Yaskawa INFORM job: X2_22-23(-90,180).JBI

/JOB
//NAME X2_22-23(-90,180)
///FOLDERNAME X2
//POS
///NPOS 121,121,119,9,0,0
///TOOL 0
///POSTYPE PULSE
///PULSE
C00000=-2000,-95440,-72516,0,38121,0
C00001=80443,-95440,-72516,46202,38121,-50067
C00002=121048,-35889,-42121,1043,37047,-65138
C00003=121557,-2539,-17456,-43794,56524,-32797
C00004=120863,2743,-10296,-44250,54945,-32361
C00005=120596,4906,-7348,-44467,54301,-32168
C00006=120755,7039,-5502,-44562,54352,-32106
C00007=120722,6457,-5983,-44548,54334,-32114
C00008=120719,6604,-4609,-44933,53775,-31814
C00009=120722,6457,-5983,-44548,54334,-32114
C00010=120988,4291,-8953,-44325,54985,-32311
C00011=121680,-993,-16157,-43855,56581,-32759
C00012=120048,-2169,-23700,-17577,56183,-40243
C00013=120438,2634,-16754,-18201,54544,-39794
C00014=120588,4602,-13901,-18464,53869,-39607
C00015=120747,6727,-12066,-18575,53869,-39539
C00016=120731,6185,-12507,-18566,53858,-39544
C00017=120727,6181,-11266,-18742,53130,-39409
C00018=120731,6185,-12507,-18566,53858,-39544
C00019=120584,4213,-15378,-18303,54543,-39732
C00020=120201,-590,-22366,-17676,56206,-40184
C00021=120684,5680,-12751,-24181,58802,-41191
C00022=120685,5691,-12742,-24181,58802,-41191
C00023=120646,5363,-16101,-23722,60533,-41605
C00024=120645,1544,-17222,-24010,59364,-41338
C00025=120685,5695,-12739,-24181,58802,-41191
C00026=120685,5705,-12730,-24145,60239,-39557
C00027=120685,5848,-12606,-24145,60236,-39557
C00028=120407,6153,-6117,-43461,53553,-40856
C00029=120685,5980,-7491,-43224,54249,-41062
C00030=120685,5834,-10671,-42343,55652,-41764
C00031=121048,-35889,-42121,1043,37047,-65138
C00032=80443,-95440,-72516,46202,38121,-50067
C00033=628,-74499,-67639,57475,89722,-72456
C00034=628,-74499,-67639,57475,89722,-72456
C00035=57022,-39792,-97587,14580,73098,-62715
C00036=77807,6055,-39746,10148,68442,-55630
C00037=79243,8316,-34713,9405,66379,-55331
C00038=80169,10516,-31635,8886,65529,-55089
C00039=80963,12031,-30280,8399,65395,-54832
C00040=80889,11723,-30556,8444,65413,-54856
C00041=80889,11351,-30020,8477,64899,-54893
C00042=80459,11155,-31041,8710,65464,-54995
C00043=79913,10174,-33131,8996,66291,-55115
C00044=78505,7891,-38206,9727,68362,-55410
C00045=77753,5785,-39720,10191,68296,-55659
C00046=79192,8060,-34680,9447,66235,-55360
C00047=82054,8043,-33590,7724,65287,-54470
C00048=82379,9432,-32364,7521,65217,-54367
C00049=82297,9081,-32674,7571,65235,-54393
C00050=82297,8847,-32336,7591,64909,-54415
C00051=80432,10909,-31095,8733,65375,-55011
C00052=79885,9924,-33187,9019,66201,-55131
C00053=78475,7632,-38265,9751,68270,-55428
C00054=83648,6461,-36170,1745,63660,-53011
C00055=83747,5652,-35361,1694,62744,-52991
C00056=84187,6753,-32863,1416,61768,-52855
C00057=81142,10477,-29433,3447,61652,-53915
C00058=80255,9791,-30406,4031,61937,-54214
C00059=80258,11096,-32246,3966,63735,-54150
C00060=57022,-39792,-97587,14580,73098,-62715
C00061=628,-74499,-67639,57475,89722,-72456
C00062=628,-74499,-67639,57475,89722,-72456
C00063=628,-74499,-67639,57475,89722,-72456
C00064=628,-74499,-67639,57475,89722,-72456
C00065=71892,-109130,-85039,20754,40171,-11669
C00066=106389,-40524,-53403,24815,61142,19479
C00067=120470,1866,-17440,30101,56195,36353
C00068=120719,2683,-16651,30153,56013,36673
C00069=120773,4699,-13768,30370,55352,36490
C00070=120564,7533,-11305,30511,55374,36401
C00071=120670,6740,-11178,30619,54915,36303
C00072=120665,6751,-9510,30988,54034,36013
C00073=120670,6740,-11178,30619,54915,36303
C00074=120615,4703,-14100,30391,55587,36492
C00075=120473,-266,-21211,29878,57224,36936
C00076=121398,-1811,-23726,17127,56782,40252
C00077=120993,2938,-16799,17744,55126,39804
C00078=120837,4887,-13955,18002,54444,39619
C00079=120627,7720,-11489,18149,54432,39528
C00080=120605,6750,-11571,18262,54010,39442
C00081=120600,6748,-9914,18499,53040,39261
C00082=120605,6750,-11571,18262,54010,39442
C00083=121150,-14,-21462,17373,56384,40085
C00084=114935,6727,-10898,18108,63991,38712
C00085=105615,-2055,-15067,38715,63232,35896
C00086=105666,5748,-4871,39423,61430,35186
C00087=115774,5149,-8950,35948,58489,37624
C00088=118188,4605,-11063,30087,58489,38356
C00089=120685,6333,-7231,42675,54657,41140
C00090=120685,6258,-8528,42321,55226,41422
C00091=120685,6198,-11659,41481,56657,42109
C00092=628,-74499,-67639,57475,89722,-72456
C00093=628,-74499,-67639,57475,89722,-72456
C00094=73729,14650,-65218,39624,99784,34982
C00095=79038,5651,-41829,36469,82879,30814
C00096=79794,8712,-36062,36285,80989,30462
C00097=80238,10863,-32413,36196,79892,30261
C00098=80449,12924,-30562,36114,79745,30290
C00099=80337,12469,-30973,36158,79803,30267
C00100=80337,11828,-30094,36241,79095,30031
C00101=80425,12177,-31517,36106,79921,30344
C00102=80141,10890,-33898,36156,80684,30490
C00103=79405,7814,-39711,36325,82587,30850
C00104=79095,5770,-41687,36447,82837,30820
C00105=79848,8834,-35915,36264,80946,30468
C00106=80509,11322,-31838,36094,79692,30298
C00107=80683,12908,-30408,36027,79574,30324
C00108=80563,12412,-30857,36075,79637,30299
C00109=80563,11846,-30077,36150,79008,30090
C00110=80446,12400,-31453,36090,79975,30369
C00111=80162,11117,-33833,36141,80739,30516
C00112=79428,8050,-39643,36311,82643,30877
C00113=80369,12305,-32773,40785,82539,30314
C00114=80366,10908,-30990,40925,81149,29769
C00115=80599,11314,-29317,40908,80419,29578
C00116=80511,11265,-29307,40945,80432,29547
C00117=80326,10673,-31042,40949,81098,29733
C00118=80329,12062,-32831,40808,82488,30278
C00119=73729,14650,-65218,39624,99784,34982
C00120=-2800,-56338,-97337,367,83074,-232
BC00000=23532,523905,788952
BC00001=125909,496171,117576
BC00002=159989,496171,117576
BC00003=146377,457946,17
BC00004=146377,457946,17
BC00005=146377,457946,17
BC00006=146377,457946,17
BC00007=146377,457946,17
BC00008=146377,457946,17
BC00009=146377,457946,17
BC00010=146377,457946,17
BC00011=146377,457946,17
BC00012=124676,474529,2658
BC00013=124676,474529,2658
BC00014=124676,474529,2658
BC00015=124676,474529,2658
BC00016=124676,474529,2658
BC00017=124676,474529,2658
BC00018=124676,474529,2658
BC00019=124676,474529,2658
BC00020=124676,474529,2658
BC00021=109348,473025,40679
BC00022=109185,468237,19665
BC00023=109120,466322,11259
BC00024=109120,466322,11259
BC00025=109120,466322,11259
BC00026=113377,463743,16288
BC00027=162486,455184,17102
BC00028=158679,453956,17
BC00029=157926,455904,17
BC00030=156043,460776,17
BC00031=159989,496171,117576
BC00032=125909,496171,117576
BC00033=97158,523229,426323
BC00034=97158,523229,1005604
BC00035=48431,468399,1061681
BC00036=65052,442237,1075139
BC00037=65052,442237,1075139
BC00038=65052,442237,1075139
BC00039=65052,442237,1075139
BC00040=65052,442237,1075139
BC00041=65052,442237,1075139
BC00042=65052,442237,1075139
BC00043=65052,442237,1075139
BC00044=65052,442237,1075139
BC00045=2261,453176,1075139
BC00046=2261,453176,1075139
BC00047=2261,453176,1075139
BC00048=2261,453176,1075139
BC00049=2261,453176,1075139
BC00050=2261,453176,1075139
BC00051=2261,453176,1075139
BC00052=2261,453176,1075139
BC00053=2261,453176,1075139
BC00054=1592,459940,1075139
BC00055=1592,454468,1075139
BC00056=1592,452279,1075139
BC00057=59392,440617,1075139
BC00058=57917,442806,1075139
BC00059=58212,448278,1075139
BC00060=48431,468399,1061681
BC00061=97158,523229,1005604
BC00062=97158,523229,842352
BC00063=97158,523229,842352
BC00064=97158,523229,1051970
BC00065=250466,483638,320114
BC00066=268157,471482,125895
BC00067=279228,463874,4352
BC00068=279439,463729,2036
BC00069=279439,463729,2036
BC00070=279439,463729,2036
BC00071=279439,463729,2036
BC00072=279439,463729,2036
BC00073=279439,463729,2036
BC00074=279439,463729,2036
BC00075=279439,463729,2036
BC00076=313684,475025,18299
BC00077=313684,475025,18299
BC00078=313684,475025,18299
BC00079=313684,475025,18299
BC00080=313684,475025,18299
BC00081=313684,475025,18299
BC00082=313684,475025,18299
BC00083=313684,475025,18299
BC00084=295059,466219,85453
BC00085=298191,460141,56261
BC00086=298191,460141,56261
BC00087=322149,463189,26141
BC00088=278371,455636,25524
BC00089=279361,453981,17
BC00090=280099,455914,17
BC00091=281944,460744,17
BC00092=97158,523229,426323
BC00093=97158,523229,1033177
BC00094=194066,506419,1075139
BC00095=165051,440056,1075139
BC00096=165051,440056,1075139
BC00097=165051,440056,1075139
BC00098=165051,440056,1075139
BC00099=165051,440056,1075139
BC00100=165051,440056,1075139
BC00101=165051,440056,1075139
BC00102=165051,440056,1075139
BC00103=165051,440056,1075139
BC00104=226024,450581,1075139
BC00105=226024,450581,1075139
BC00106=226024,450581,1075139
BC00107=226024,450581,1075139
BC00108=226024,450581,1075139
BC00109=226024,450581,1075139
BC00110=226024,450581,1075139
BC00111=226024,450581,1075139
BC00112=226024,450581,1075139
BC00113=238899,457644,1075139
BC00114=239227,452207,1075139
BC00115=239359,450033,1075139
BC00116=172415,438485,1075139
BC00117=172284,440660,1075139
BC00118=171955,446096,1075139
BC00119=194066,506419,1075139
BC00120=194066,523905,1075139
EC00000=798156,-1296783
EC00001=798156,-1296783
EC00002=798156,-1296783
EC00003=798156,-1296783
EC00004=798156,-1296783
EC00005=798156,-1296783
EC00006=798156,-1296783
EC00007=798156,-1296783
EC00008=798156,-1296783
EC00009=798156,-1296783
EC00010=798156,-1296783
EC00011=798156,-1296783
EC00012=798156,-1296783
EC00013=798156,-1296783
EC00014=798156,-1296783
EC00015=798156,-1296783
EC00016=798156,-1296783
EC00017=798156,-1296783
EC00018=798156,-1296783
EC00019=798156,-1296783
EC00020=798156,-1296783
EC00021=798156,-1296783
EC00022=798156,-1296783
EC00023=798156,-1296783
EC00024=798156,-1296783
EC00025=798156,-1296783
EC00026=798156,-1296783
EC00027=798156,-1296783
EC00028=798156,-1296783
EC00029=798156,-1296783
EC00030=798156,-1296783
EC00031=798156,-1296783
EC00032=798156,-1296783
EC00033=798156,-1296783
EC00034=798156,-1296783
EC00035=798156,-1296783
EC00036=798156,-1296783
EC00037=798156,-1296783
EC00038=798156,-1296783
EC00039=798156,-1296783
EC00040=798156,-1296783
EC00041=798156,-1296783
EC00042=798156,-1296783
EC00043=798156,-1296783
EC00044=798156,-1296783
EC00045=798156,-1296783
EC00046=798156,-1296783
EC00047=798156,-1296783
EC00048=798156,-1296783
EC00049=798156,-1296783
EC00050=798156,-1296783
EC00051=798156,-1296783
EC00052=798156,-1296783
EC00053=798156,-1296783
EC00054=798156,-1296783
EC00055=798156,-1296783
EC00056=798156,-1296783
EC00057=798156,-1296783
EC00058=798156,-1296783
EC00059=798156,-1296783
EC00060=859390,-983133
EC00061=868219,-545682
EC00062=798156,-183832
EC00063=798156,-183832
EC00064=798156,-183832
EC00065=798156,-183832
EC00066=798156,-183832
EC00067=798156,-183832
EC00068=798156,-183832
EC00069=798156,-183832
EC00070=798156,-183832
EC00071=798156,-183832
EC00072=798156,-183832
EC00073=798156,-183832
EC00074=798156,-183832
EC00075=798156,-183832
EC00076=798156,-183832
EC00077=798156,-183832
EC00078=798156,-183832
EC00079=798156,-183832
EC00080=798156,-183832
EC00081=798156,-183832
EC00082=798156,-183832
EC00083=798156,-183832
EC00084=798156,-183832
EC00085=798156,-183832
EC00086=798156,-183832
EC00087=798156,-183832
EC00088=798156,-183832
EC00089=798156,-183832
EC00090=798156,-183832
EC00091=798156,-183832
EC00092=798156,-183832
EC00093=798156,-183832
EC00094=798156,-183832
EC00095=798156,-183832
EC00096=798156,-183832
EC00097=798156,-183832
EC00098=798156,-183832
EC00099=798156,-183832
EC00100=798156,-183832
EC00101=798156,-183832
EC00102=798156,-183832
EC00103=798156,-183832
EC00104=798156,-183832
EC00105=798156,-183832
EC00106=798156,-183832
EC00107=798156,-183832
EC00108=798156,-183832
EC00109=798156,-183832
EC00110=798156,-183832
EC00111=798156,-183832
EC00112=798156,-183832
EC00113=798156,-183832
EC00114=798156,-183832
EC00115=798156,-183832
EC00116=798156,-183832
EC00117=798156,-183832
EC00118=798156,-183832
///POSTYPE BASE
///RECTAN
///RCONF 0,0,0,0,1,0,0,0,0,0,0,0,0,0,0,0,0,0,0,0,0,0,0,0
P00006=2.006,1.622,-0.565,0.0000,0.0000,0.0000
P00021=0.073,2.058,-0.109,0.0000,0.0000,0.0000
P00022=2.006,1.622,-0.565,0.0000,0.0000,0.0000
///RCONF 0,0,0,0,0,0,0,0,0,0,0,0,0,0,0,0,0,0,0,0,0,0,0,0
P00023=-2.957,-4.083,2.762,0.0000,0.0000,0.0000
P00024=-1.466,-0.226,-0.419,0.0000,0.0000,0.0000
P00025=3.643,0.007,-2.585,0.0000,0.0000,0.0000
P00026=2.644,0.055,-2.583,0.0000,0.0000,0.0000
P00027=2.278,0.099,-4.210,0.0000,0.0000,0.0000
P00028=-1.778,-0.182,-2.050,0.0000,0.0000,0.0000
//INST
///DATE 2024/12/18 14:18
///ATTR SC,RW
///GROUP1 RB1,BS1
///GROUP2 ST1
NOP
'X2_22-23(-90,180)
MOVJ C00000 BC00000 VJ=100.00  +MOVJ EC00000 VJ=100.00
MOVJ C00001 BC00001 VJ=100.00  +MOVJ EC00001 VJ=100.00
MOVJ C00002 BC00002 VJ=100.00  +MOVJ EC00002 VJ=100.00
'Path S4216
SFTOF3D
MOVJ C00003 BC00003 VJ=100.00  +MOVJ EC00003 VJ=100.00
MOVL C00004 BC00004 V=800.0  +MOVJ EC00004 VJ=100.00
SMOVL C00005 BC00005 V=166.7  +MOVJ EC00005
SREFP 3 C00006 BC00006  +REFP EC00006
CALL JOB:SEARCH-R1-S13D
SET P022 P006
SFTON3D P022
SMOVL C00007 BC00007 V=166.7  +MOVJ EC00007
SREFP 3 C00008 BC00008  +REFP EC00008
CALL JOB:SEARCH-R1-S13D
SET P022 P006
SFTON3D P022
SMOVL C00009 BC00009 V=166.7  +MOVJ EC00009
MOVL C00010 BC00010 V=800.0  +MOVJ EC00010 VJ=100.00
MOVL C00011 BC00011 V=1000.0  +MOVJ EC00011 VJ=100.00
'EndPath S4216
'Path S3525
SFTOF3D
MOVJ C00012 BC00012 VJ=100.00  +MOVJ EC00012 VJ=100.00
MOVL C00013 BC00013 V=800.0  +MOVJ EC00013 VJ=100.00
SMOVL C00014 BC00014 V=166.7  +MOVJ EC00014
SREFP 3 C00015 BC00015  +REFP EC00015
CALL JOB:SEARCH-R1-S13D
SET P021 P006
SFTON3D P021
SMOVL C00016 BC00016 V=166.7  +MOVJ EC00016
SREFP 3 C00017 BC00017  +REFP EC00017
CALL JOB:SEARCH-R1-S13D
SET P021 P006
SFTON3D P021
SMOVL C00018 BC00018 V=166.7  +MOVJ EC00018
MOVL C00019 BC00019 V=800.0  +MOVJ EC00019 VJ=100.00
MOVL C00020 BC00020 V=1000.0  +MOVJ EC00020 VJ=100.00
'EndPath S3525
'Path W3526
SFTOF3D
SFTON3D P021
MOVJ C00021 BC00021 VJ=100.00  +MOVJ EC00021 VJ=100.00
SMOVL C00022 BC00022 V=800.0  +MOVJ EC00022
REFP 1 RB1 C00023 BC00023
REFP 2 RB1 C00024 BC00024
SMOVL C00025 BC00025 V=166.7 PL=0  +MOVJ EC00023
MACRO1 MJ#(0) ARGF18
ARCON
SMOVL C00026 BC00026 V=8.3  +MOVJ EC00024
SFTON3D P022
SMOVL C00027 BC00027 V=8.3  +MOVJ EC00025
SMOVL C00028 BC00028 V=8.3  +MOVJ EC00026
ARCOF
SMOVL C00029 BC00029 V=800.0  +MOVJ EC00027
SMOVL C00030 BC00030 V=1000.0  +MOVJ EC00028
SFTOF3D
'EndPath W3526
MOVJ C00031 BC00031 VJ=100.00  +MOVJ EC00029 VJ=100.00
MOVJ C00032 BC00032 VJ=100.00  +MOVJ EC00030 VJ=100.00
MOVJ C00033 BC00033 VJ=100.00  +MOVJ EC00031 VJ=100.00
'R-L Trip
MOVJ C00034 BC00034 VJ=100.00  +MOVJ EC00032 VJ=100.00
CALL JOB:CLEAN-R1_KM_NEW
MOVJ C00035 BC00035 VJ=100.00  +MOVJ EC00033 VJ=100.00
'Path S4217
SFTOF3D
MOVJ C00036 BC00036 VJ=100.00  +MOVJ EC00034 VJ=100.00
MOVL C00037 BC00037 V=800.0  +MOVJ EC00035 VJ=100.00
SMOVL C00038 BC00038 V=166.7  +MOVJ EC00036
SREFP 3 C00039 BC00039  +REFP EC00037
CALL JOB:SEARCH-R1-S13D
SET P024 P006
SFTON3D P024
SMOVL C00040 BC00040 V=166.7  +MOVJ EC00038
SREFP 3 C00041 BC00041  +REFP EC00039
CALL JOB:SEARCH-R1-S13D
SET P024 P006
SFTON3D P024
SMOVL C00042 BC00042 V=166.7  +MOVJ EC00040
MOVL C00043 BC00043 V=800.0  +MOVJ EC00041 VJ=100.00
MOVL C00044 BC00044 V=1000.0  +MOVJ EC00042 VJ=100.00
'EndPath S4217
'Path S3527
SFTOF3D
MOVJ C00045 BC00045 VJ=100.00  +MOVJ EC00043 VJ=100.00
MOVL C00046 BC00046 V=800.0  +MOVJ EC00044 VJ=100.00
SMOVL C00047 BC00047 V=166.7  +MOVJ EC00045
SREFP 3 C00048 BC00048  +REFP EC00046
CALL JOB:SEARCH-R1-S13D
SET P023 P006
SFTON3D P023
SMOVL C00049 BC00049 V=166.7  +MOVJ EC00047
SREFP 3 C00050 BC00050  +REFP EC00048
CALL JOB:SEARCH-R1-S13D
SET P023 P006
SFTON3D P023
SMOVL C00051 BC00051 V=166.7  +MOVJ EC00049
MOVL C00052 BC00052 V=800.0  +MOVJ EC00050 VJ=100.00
MOVL C00053 BC00053 V=1000.0  +MOVJ EC00051 VJ=100.00
'EndPath S3527
'Path W4169
SFTOF3D
SFTON3D P023
MOVJ C00054 BC00054 VJ=100.00  +MOVJ EC00052 VJ=100.00
SMOVL C00055 BC00055 V=666.7  +MOVJ EC00053
SMOVL C00056 BC00056 V=166.7 PL=0  +MOVJ EC00054
ARCON
SFTON3D P024
SMOVL C00057 BC00057 V=8.3  +MOVJ EC00055
ARCOF
SMOVL C00058 BC00058 V=800.0  +MOVJ EC00056
SMOVL C00059 BC00059 V=1000.0  +MOVJ EC00057
SFTOF3D
'EndPath W4169
MOVJ C00060 BC00060 VJ=100.00  +MOVJ EC00058 VJ=100.00
MOVJ C00061 BC00061 VJ=100.00  +MOVJ EC00059 VJ=100.00
MOVJ C00062 BC00062 VJ=100.00  +MOVJ EC00060 VJ=100.00
MOVJ C00063 BC00063 VJ=100.00  +MOVJ EC00061 VJ=100.00
MOVJ C00064 BC00064 VJ=100.00  +MOVJ EC00062 VJ=100.00
'Path S4218
SFTOF3D
CALL JOB:CLEAN-R1_KM_NEW
MOVJ C00065 BC00065 VJ=100.00  +MOVJ EC00063 VJ=100.00
MOVJ C00066 BC00066 VJ=100.00  +MOVJ EC00064 VJ=100.00
MOVL C00067 BC00067 V=1000.0  +MOVJ EC00065 VJ=100.00
MOVL C00068 BC00068 V=800.0  +MOVJ EC00066 VJ=100.00
SMOVL C00069 BC00069 V=166.7  +MOVJ EC00067
SREFP 3 C00070 BC00070  +REFP EC00068
CALL JOB:SEARCH-R1-S13D
SET P026 P006
SFTON3D P026
SMOVL C00071 BC00071 V=166.7  +MOVJ EC00069
SREFP 3 C00072 BC00072  +REFP EC00070
CALL JOB:SEARCH-R1-S13D
SET P026 P006
SFTON3D P026
SMOVL C00073 BC00073 V=166.7  +MOVJ EC00071
MOVL C00074 BC00074 V=800.0  +MOVJ EC00072 VJ=100.00
MOVL C00075 BC00075 V=1000.0  +MOVJ EC00073 VJ=100.00
'EndPath S4218
'Path S3529
SFTOF3D
MOVJ C00076 BC00076 VJ=100.00  +MOVJ EC00074 VJ=100.00
MOVL C00077 BC00077 V=800.0  +MOVJ EC00075 VJ=100.00
SMOVL C00078 BC00078 V=166.7  +MOVJ EC00076
SREFP 3 C00079 BC00079  +REFP EC00077
CALL JOB:SEARCH-R1-S13D
SET P025 P006
SFTON3D P025
SMOVL C00080 BC00080 V=166.7  +MOVJ EC00078
SREFP 3 C00081 BC00081  +REFP EC00079
CALL JOB:SEARCH-R1-S13D
SET P025 P006
SFTON3D P025
SMOVL C00082 BC00082 V=166.7  +MOVJ EC00080
MOVL C00083 BC00083 V=1000.0  +MOVJ EC00081 VJ=100.00
'EndPath S3529
'Path W3530
SFTOF3D
SFTON3D P025
MOVJ C00084 BC00084 VJ=100.00  +MOVJ EC00082 VJ=100.00
SMOVL C00085 BC00085 V=800.0  +MOVJ EC00083
SMOVL C00086 BC00086 V=166.7 PL=0  +MOVJ EC00084
ARCON
SMOVL C00087 BC00087 V=8.3  +MOVJ EC00085
SFTON3D P026
SMOVL C00088 BC00088 V=8.3  +MOVJ EC00086
SMOVL C00089 BC00089 V=8.3  +MOVJ EC00087
ARCOF
SMOVL C00090 BC00090 V=800.0  +MOVJ EC00088
SMOVL C00091 BC00091 V=1000.0  +MOVJ EC00089
SFTOF3D
'EndPath W3530
'L-R Trip
MOVJ C00092 BC00092 VJ=100.00  +MOVJ EC00090 VJ=100.00
MOVJ C00093 BC00093 VJ=100.00  +MOVJ EC00091 VJ=100.00
CALL JOB:CLEAN-R1_KM_NEW
MOVJ C00094 BC00094 VJ=100.00  +MOVJ EC00092 VJ=100.00
'Path S4219
SFTOF3D
MOVJ C00095 BC00095 VJ=100.00  +MOVJ EC00093 VJ=100.00
MOVL C00096 BC00096 V=800.0  +MOVJ EC00094 VJ=100.00
SMOVL C00097 BC00097 V=166.7  +MOVJ EC00095
SREFP 3 C00098 BC00098  +REFP EC00096
CALL JOB:SEARCH-R1-S13D
SET P028 P006
SFTON3D P028
SMOVL C00099 BC00099 V=166.7  +MOVJ EC00097
SREFP 3 C00100 BC00100  +REFP EC00098
CALL JOB:SEARCH-R1-S13D
SET P028 P006
SFTON3D P028
SMOVL C00101 BC00101 V=166.7  +MOVJ EC00099
MOVL C00102 BC00102 V=800.0  +MOVJ EC00100 VJ=100.00
MOVL C00103 BC00103 V=1000.0  +MOVJ EC00101 VJ=100.00
'EndPath S4219
'Path S3531
SFTOF3D
MOVJ C00104 BC00104 VJ=100.00  +MOVJ EC00102 VJ=100.00
MOVL C00105 BC00105 V=800.0  +MOVJ EC00103 VJ=100.00
SMOVL C00106 BC00106 V=166.7  +MOVJ EC00104
SREFP 3 C00107 BC00107  +REFP EC00105
CALL JOB:SEARCH-R1-S13D
SET P027 P006
SFTON3D P027
SMOVL C00108 BC00108 V=166.7  +MOVJ EC00106
SREFP 3 C00109 BC00109  +REFP EC00107
CALL JOB:SEARCH-R1-S13D
SET P027 P006
SFTON3D P027
SMOVL C00110 BC00110 V=166.7  +MOVJ EC00108
MOVL C00111 BC00111 V=800.0  +MOVJ EC00109 VJ=100.00
MOVL C00112 BC00112 V=1000.0  +MOVJ EC00110 VJ=100.00
'EndPath S3531
'Path W4177
SFTOF3D
SFTON3D P027
MOVJ C00113 BC00113 VJ=100.00  +MOVJ EC00111 VJ=100.00
SMOVL C00114 BC00114 V=800.0  +MOVJ EC00112
SMOVL C00115 BC00115 V=150.0 PL=0  +MOVJ EC00113
ARCON
SFTON3D P028
SMOVL C00116 BC00116 V=8.3  +MOVJ EC00114
ARCOF
SMOVL C00117 BC00117 V=800.0  +MOVJ EC00115
SMOVL C00118 BC00118 V=1000.0  +MOVJ EC00116
SFTOF3D
'EndPath W4177
MOVJ C00119 BC00119 VJ=100.00  +MOVJ EC00117 VJ=100.00
MOVJ C00120 BC00120 VJ=100.00  +MOVJ EC00118 VJ=100.00
END
